// TIA Portal V20 export
// export: Created 2025-12-01T14:57:05.2668309Z, ExportSetting None, DisplayName Totally Integrated Automation Portal, DisplayVersion V20 Update 3, DisplayName TIA Portal Openness, DisplayVersion V20 Update 3, DisplayName TIA Portal Version Control Interface, DisplayVersion V20 Update 3, DisplayName STEP 7 Professional, DisplayVersion V20 Update 3, DisplayName STEP 7 Safety, DisplayVersion V20 Update 2, DisplayName WinCC Basic/Comfort/Advanced, DisplayVersion V20 Update 3, DisplayName WinCC Professional, DisplayVersion V20 Update 3, DisplayName WinCC Unified, DisplayVersion V20 Update 3
FUNCTION "FC777_TipoCajaPlastico_EnMesa" : Void   // FC777, STL
TITLE = Informacion del tipo de Caja en la Mesa
{ S7_Optimized_Access := 'FALSE' }
AUTHOR : TRACKING
NAME : 20130301
VERSION : 3.0
// stored: AutoNumber false
   VAR_INPUT
      Mesa : UInt;   // Numero de Mesa
   END_VAR
   VAR_OUTPUT
      DosCajas : Bool;   // Hay dos Cajas en la Mesa
      CajaPeque_UT01 : Bool;   // Caja Primera Pequeña
      CajaPeque_UT02 : Bool;   // Caja Segunda Pequeña
   END_VAR
   VAR_TEMP
      NumeroUT : UInt;
   END_VAR
BEGIN

NETWORK
TITLE = Inicialializar
////////////////////////////////////////////////////////////////////////////
// --- Inicializar Variables

      SET;
      R     #DosCajas;
      R     #CajaPeque_UT01;
      R     #CajaPeque_UT02;



NETWORK
TITLE = Calculo de Activacion
////////////////////////////////////////////////////////////////////////////
// --- Ver si hay UT's en la Mesa

      L     "DB810_ColasMesas".Colas[#Mesa].UT_PrimeraMesa;  // Si no hay UT's
      T     #NumeroUT;

      L     #NumeroUT;
      L     0;
      ==I;
      JC    Final;


////////////////////////////////////////////////////////////////////////////
// --- Mirar el Tipo de Caja de la Primera UT

      L     "DB812_UTs_Control".UT[#NumeroUT].TipoCarga;
      L     10;
      /I;
      L     10;  // CajaPequeña (3x)
      ==I;
      S     #CajaPeque_UT01;


////////////////////////////////////////////////////////////////////////////
// --- Mirar el Tipo de Caja de la Segunda UT, si Hay
// ---

      L     "DB812_UTs_Control".UT[#NumeroUT].UT_SiguienteMesa;
      T     #NumeroUT;

      L     #NumeroUT;
      L     0;
      ==I;
      JC    Final;  // Quedan UT's en la Mesa ?

      SET;
      S     #DosCajas;  // Hay dos cajas en la Mesa

// Nota: Siempre deberia ser pequeña, pero comprobamos

      L     "DB812_UTs_Control".UT[#NumeroUT].TipoCarga;
      L     10;
      /I;
      L     10;  // CajaPequeña (3x)
      ==I;
      S     #CajaPeque_UT02;



NETWORK
TITLE = Final de la Funcion
////////////////////////////////////////////////////////////////////////////
// --- Final de la Funcion
Final:NOP   0;

END_FUNCTION
